// TIA Portal V18 export
// export: Created 2026-01-09T11:32:03.8711545Z, ExportSetting WithDefaults, DisplayName Totally Integrated Automation Portal, DisplayVersion V18 Update 5, DisplayName TIA Portal Openness, DisplayVersion V18 Update 5, DisplayName TIA Portal Teamcenter Gateway, DisplayVersion V18, DisplayName TIA Portal Version Control Interface, DisplayVersion V18, DisplayName SINAMICS Startdrive Advanced, DisplayVersion V18 SP2 Update 1, DisplayName SINAMICS Startdrive G110M, G120, G120C, G120D, G120P, G115D, DisplayVersion V18 SP2 Update 1, DisplayName SINAMICS Startdrive G130, G150, S120, S150, SINAMICS MV, S210, G220, S200, DisplayVersion V18 SP2 Update 1, DisplayName STEP 7 Professional, DisplayVersion V18 Update 5, DisplayName STEP 7 Safety, DisplayVersion V18, DisplayName WinCC Professional, DisplayVersion V18 Update 5
TagTable "ST_Initial"
  ST_InitialRunning : Bool  (%DB[ST_SysDBNum].DBX70.1, CPU S71500-2PN_TP700, 1 s)
  ST_InitialRunning[1] : Bool  (%DB[ST_PMDBNum].DBX0.2, CPU S71500-2PN_TP700, 1 s)
  ST_InitialRunning[10] : Bool  (%DB[ST_PMDBNum].DBX180.2, CPU S71500-2PN_TP700, 1 s)
  ST_InitialRunning[11] : Bool  (%DB[ST_PMDBNum].DBX200.2, CPU S71500-2PN_TP700, 1 s)
  ST_InitialRunning[12] : Bool  (%DB[ST_PMDBNum].DBX220.2, CPU S71500-2PN_TP700, 1 s)
  ST_InitialRunning[13] : Bool  (%DB[ST_PMDBNum].DBX240.2, CPU S71500-2PN_TP700, 1 s)
  ST_InitialRunning[14] : Bool  (%DB[ST_PMDBNum].DBX260.2, CPU S71500-2PN_TP700, 1 s)
  ST_InitialRunning[15] : Bool  (%DB[ST_PMDBNum].DBX280.2, CPU S71500-2PN_TP700, 1 s)
  ST_InitialRunning[2] : Bool  (%DB[ST_PMDBNum].DBX20.2, CPU S71500-2PN_TP700, 1 s)
  ST_InitialRunning[3] : Bool  (%DB[ST_PMDBNum].DBX40.2, CPU S71500-2PN_TP700, 1 s)
  ST_InitialRunning[4] : Bool  (%DB[ST_PMDBNum].DBX60.2, CPU S71500-2PN_TP700, 1 s)
  ST_InitialRunning[5] : Bool  (%DB[ST_PMDBNum].DBX80.2, CPU S71500-2PN_TP700, 1 s)
  ST_InitialRunning[6] : Bool  (%DB[ST_PMDBNum].DBX100.2, CPU S71500-2PN_TP700, 1 s)
  ST_InitialRunning[7] : Bool  (%DB[ST_PMDBNum].DBX120.2, CPU S71500-2PN_TP700, 1 s)
  ST_InitialRunning[8] : Bool  (%DB[ST_PMDBNum].DBX140.2, CPU S71500-2PN_TP700, 1 s)
  ST_InitialRunning[9] : Bool  (%DB[ST_PMDBNum].DBX160.2, CPU S71500-2PN_TP700, 1 s)
  ST_SetInitial : Bool  (%DB[ST_SysDBNum].DBX70.0, CPU S71500-2PN_TP700, 1 s)
  ST_SetInitial[1] : Bool  (%DB[ST_PMDBNum].DBX0.1, CPU S71500-2PN_TP700, 1 s)
  ST_SetInitial[10] : Bool  (%DB[ST_PMDBNum].DBX180.1, CPU S71500-2PN_TP700, 1 s)
  ST_SetInitial[11] : Bool  (%DB[ST_PMDBNum].DBX200.1, CPU S71500-2PN_TP700, 1 s)
  ST_SetInitial[12] : Bool  (%DB[ST_PMDBNum].DBX220.1, CPU S71500-2PN_TP700, 1 s)
  ST_SetInitial[13] : Bool  (%DB[ST_PMDBNum].DBX240.1, CPU S71500-2PN_TP700, 1 s)
  ST_SetInitial[14] : Bool  (%DB[ST_PMDBNum].DBX260.1, CPU S71500-2PN_TP700, 1 s)
  ST_SetInitial[15] : Bool  (%DB[ST_PMDBNum].DBX280.1, CPU S71500-2PN_TP700, 1 s)
  ST_SetInitial[2] : Bool  (%DB[ST_PMDBNum].DBX20.1, CPU S71500-2PN_TP700, 1 s)
  ST_SetInitial[3] : Bool  (%DB[ST_PMDBNum].DBX40.1, CPU S71500-2PN_TP700, 1 s)
  ST_SetInitial[4] : Bool  (%DB[ST_PMDBNum].DBX60.1, CPU S71500-2PN_TP700, 1 s)
  ST_SetInitial[5] : Bool  (%DB[ST_PMDBNum].DBX80.1, CPU S71500-2PN_TP700, 1 s)
  ST_SetInitial[6] : Bool  (%DB[ST_PMDBNum].DBX100.1, CPU S71500-2PN_TP700, 1 s)
  ST_SetInitial[7] : Bool  (%DB[ST_PMDBNum].DBX120.1, CPU S71500-2PN_TP700, 1 s)
  ST_SetInitial[8] : Bool  (%DB[ST_PMDBNum].DBX140.1, CPU S71500-2PN_TP700, 1 s)
  ST_SetInitial[9] : Bool  (%DB[ST_PMDBNum].DBX160.1, CPU S71500-2PN_TP700, 1 s)
  ST_SetInitial[16] : Bool  (%DB[ST_PMDBNum].DBX300.1, CPU S71500-2PN_TP700, 1 s)
  ST_InitialRunning[16] : Bool  (%DB[ST_PMDBNum].DBX300.2, CPU S71500-2PN_TP700, 1 s)
  ST10_Sys_Initial_OK : Bool  (%DB[ST_SysDBNum].DBX70.2, CPU S71500-2PN_TP700, 1 s)
  ST_InitialRunning[25] : Bool  (%DB[ST_PMDBNum].DBX480.2, CPU S71500-2PN_TP700, 1 s)
  ST_InitialRunning[24] : Bool  (%DB[ST_PMDBNum].DBX460.2, CPU S71500-2PN_TP700, 1 s)
  ST_InitialRunning[23] : Bool  (%DB[ST_PMDBNum].DBX440.2, CPU S71500-2PN_TP700, 1 s)
  ST_InitialRunning[22] : Bool  (%DB[ST_PMDBNum].DBX420.2, CPU S71500-2PN_TP700, 1 s)
  ST_InitialRunning[21] : Bool  (%DB[ST_PMDBNum].DBX400.2, CPU S71500-2PN_TP700, 1 s)
  ST_InitialRunning[20] : Bool  (%DB[ST_PMDBNum].DBX380.2, CPU S71500-2PN_TP700, 1 s)
  ST_InitialRunning[19] : Bool  (%DB[ST_PMDBNum].DBX360.2, CPU S71500-2PN_TP700, 1 s)
  ST_InitialRunning[18] : Bool  (%DB[ST_PMDBNum].DBX340.2, CPU S71500-2PN_TP700, 1 s)
  ST_InitialRunning[17] : Bool  (%DB[ST_PMDBNum].DBX320.2, CPU S71500-2PN_TP700, 1 s)
  ST_InitialRunning[30] : Bool  (%DB[ST_PMDBNum].DBX580.2, CPU S71500-2PN_TP700, 1 s)
  ST_InitialRunning[29] : Bool  (%DB[ST_PMDBNum].DBX560.2, CPU S71500-2PN_TP700, 1 s)
  ST_InitialRunning[28] : Bool  (%DB[ST_PMDBNum].DBX540.2, CPU S71500-2PN_TP700, 1 s)
  ST_InitialRunning[27] : Bool  (%DB[ST_PMDBNum].DBX520.2, CPU S71500-2PN_TP700, 1 s)
  ST_InitialRunning[26] : Bool  (%DB[ST_PMDBNum].DBX500.2, CPU S71500-2PN_TP700, 1 s)
  ST_SetInitial[17] : Bool  (%DB[ST_PMDBNum].DBX320.1, CPU S71500-2PN_TP700, 1 s)
  ST_SetInitial[18] : Bool  (%DB[ST_PMDBNum].DBX340.1, CPU S71500-2PN_TP700, 1 s)
  ST_SetInitial[19] : Bool  (%DB[ST_PMDBNum].DBX360.1, CPU S71500-2PN_TP700, 1 s)
  ST_SetInitial[20] : Bool  (%DB[ST_PMDBNum].DBX380.1, CPU S71500-2PN_TP700, 1 s)
  ST_SetInitial[21] : Bool  (%DB[ST_PMDBNum].DBX400.1, CPU S71500-2PN_TP700, 1 s)
  ST_SetInitial[22] : Bool  (%DB[ST_PMDBNum].DBX420.1, CPU S71500-2PN_TP700, 1 s)
  ST_SetInitial[23] : Bool  (%DB[ST_PMDBNum].DBX440.1, CPU S71500-2PN_TP700, 1 s)
  ST_SetInitial[24] : Bool  (%DB[ST_PMDBNum].DBX460.1, CPU S71500-2PN_TP700, 1 s)
  ST_SetInitial[25] : Bool  (%DB[ST_PMDBNum].DBX480.1, CPU S71500-2PN_TP700, 1 s)
  ST_SetInitial[26] : Bool  (%DB[ST_PMDBNum].DBX500.1, CPU S71500-2PN_TP700, 1 s)
  ST_SetInitial[27] : Bool  (%DB[ST_PMDBNum].DBX520.1, CPU S71500-2PN_TP700, 1 s)
  ST_SetInitial[28] : Bool  (%DB[ST_PMDBNum].DBX540.1, CPU S71500-2PN_TP700, 1 s)
  ST_SetInitial[29] : Bool  (%DB[ST_PMDBNum].DBX560.1, CPU S71500-2PN_TP700, 1 s)
  ST_SetInitial[30] : Bool  (%DB[ST_PMDBNum].DBX580.1, CPU S71500-2PN_TP700, 1 s)
